// TwinCAT 3 PLC project Untitled1
// ProgramVersion: 3.1.4024.0
// libraries:
//   Tc2_MC2, * (Beckhoff Automation GmbH)
//   Tc2_Standard, * (Beckhoff Automation GmbH)
//   Tc2_System, * (Beckhoff Automation GmbH)
//   Tc3_Module, * (Beckhoff Automation GmbH)
// project tree:
//   Error/DUTs/ E_ErrorPriority.TcDUT, ST_Error.TcDUT
//   Error/GVLs/ Param_Error.TcGVL
//   Error/POUs/ F_ClearError.TcPOU, F_ResetErrorList.TcPOU
//   PermIntlk/PermIntlk/ FB_PermIntlk.TcPOU, GVL_PermIntlk.TcGVL, ITF_PermIntlk.TcIO, Param_PermIntlk.TcGVL, ST_PermIntlkIndex.TcDUT
//   / PlcTask.TcTTO
//   POUs/ MAIN.TcPOU (not stored)
//   Servo/DUTs/ E_ServoTypeMoves.TcDUT, ST_ServoAxisMove.TcDUT (not stored), ST_ServoConfiguration.TcDUT (not stored), ST_ServoInterlocks.TcDUT, ST_ServoMove.TcDUT, ST_ServoStatus.TcDUT
//   Servo/ FB_Servo.TcPOU (not stored), ITF_Servo.TcIO (not stored)
//   Servo/GVLs/ Param_Servo.TcGVL
// real-time tasks:
//   TASK PlcTask: cycle T#10ms, priority 20, ADS port 350
// motion (NC):
//   TASK NC-Task 1 SAF: cycle T#2ms, priority 4, ADS port 501
//   TASK NC-Task 1 SVB: cycle T#10ms, priority 8, ADS port 511
//   AXIS Axis 1 (id 1)
//     OtherSettings: AllowMotionCmdToSlave=true
//     encoder EncType=1
//     drive DrvType=5
//       Analog: TorqueSetpointScale=10, ScaleFactorActTorque=0.1
//       TimeComp: TaskDelayCycles=1
//     controller CtrType=1
//       CtrPara: PriorControlFactor=1
//         Observer: BandWidth=20
// variable links:
//   Untitled1/Untitled1 Instance <-> NC-Task 1 SAF/Axes/Axis 1
//     PlcTask Inputs/MAIN.Servo.Axis.NcToPlc <-> Outputs/ToPlc
//     PlcTask Outputs/MAIN.Servo.Axis.PlcToNc <-> Inputs/FromPlc

CONFIGURATION Untitled1
    RESOURCE PLC ON TwinCAT3
        TASK PlcTask(INTERVAL := T#10ms, PRIORITY := 20);
        PROGRAM MAIN WITH PlcTask : MAIN;
    END_RESOURCE
END_CONFIGURATION

// ---- Error/DUTs/E_ErrorPriority.TcDUT
{attribute 'qualified_only'}
{attribute 'strict'}
TYPE E_ErrorPriority :
(
	Diagnostic := 0,
	Low := 1,
	Medium := 2,
	High := 3,
	Critical := 4
);
END_TYPE

// ---- Error/DUTs/ST_Error.TcDUT
TYPE ST_Error :
STRUCT
	Active : BOOL := FALSE;
	Label : STRING(Param_Error.LABEL_LEN);
	Message : STRING(Param_Error.MESSAGE_LEN);
	Priority : E_ErrorPriority := E_ErrorPriority.Diagnostic;
END_STRUCT
END_TYPE

// ---- PermIntlk/PermIntlk/ST_PermIntlkIndex.TcDUT
TYPE ST_PermIntlkIndex :
STRUCT
	Condition : BOOL := TRUE;
	Description : STRING(Param_PermIntlk.DESCRIPTION_LEN);
END_STRUCT
END_TYPE

// ---- Servo/DUTs/E_ServoTypeMoves.TcDUT
{attribute 'qualified_only'}
{attribute 'strict'}
TYPE E_ServoTypeMoves :
(
	AbsoluteMove := 0,
	RelativeMove := 1,
	VelocityMove := 2,
	DynamicGear  := 3
);
END_TYPE

// ---- Servo/DUTs/ST_ServoInterlocks.TcDUT
TYPE ST_ServoInterlocks :
STRUCT
	Move_Positive : BOOL;
	Move_Negative : BOOL;
	SafetyOk     : BOOL;
	
END_STRUCT
END_TYPE

// ---- Servo/DUTs/ST_ServoMove.TcDUT
TYPE ST_ServoMove :
STRUCT
	Name : STRING(Param_Servo.DESCRIPTION_LEN) := 'Actuator'; //Name visualized on UI
	AdvanceFeedback_Used : BOOL;      //TRUE if advanced state feedback is used  
	RetractFeedback_Used  : BOOL;      //TRUE if retracted state feedback is used  
	AdvanceFeedbackTimeoutError : TIME; // How long we wait to see advanced feedback before we raise timeout error; 0 if not used
	RetractFeedbackTimeoutError : TIME; // How long we wait to see retracted feedback before we raise timeout error; 0 if not used
	SimFeedback_Advance_TimeElapsed : TIME; //If we do not use Advanced Feedback, serves as simulation delay after Advance Output is Set
	SimFeedback_Retract_TimeElapsed : TIME; //If we do not use Retracted Feedback, serves as simulation delay after Advance Output is Set
END_STRUCT
END_TYPE

// ---- Servo/DUTs/ST_ServoStatus.TcDUT
TYPE ST_ServoStatus :
STRUCT
	
	//Status : AXIS_REF.Status;

END_STRUCT
END_TYPE

// ---- Error/GVLs/Param_Error.TcGVL
{attribute 'qualified_only'}
VAR_GLOBAL CONSTANT
	LABEL_LEN : USINT := 40;
	MESSAGE_LEN : USINT := 255;
END_VAR

// ---- PermIntlk/PermIntlk/GVL_PermIntlk.TcGVL
{attribute 'qualified_only'}
{attribute 'global_init_slot' := '49991'}
VAR_GLOBAL CONSTANT
	EMPTY_INDICES : ARRAY[0..(Param_PermIntlk.ARRAY_SIZE-1)] OF ST_PermIntlkIndex := [(Param_Permintlk.ARRAY_SIZE -1)((Condition := TRUE, Description := ''))];
END_VAR

// ---- PermIntlk/PermIntlk/Param_PermIntlk.TcGVL
{attribute 'qualified_only'}
{attribute 'global_init_slot := '49990'}
VAR_GLOBAL CONSTANT
	ARRAY_SIZE : USINT := 16;
	DESCRIPTION_LEN : USINT := 40;
	MESSAGE_LEN : USINT := 127;
END_VAR

// ---- Servo/GVLs/Param_Servo.TcGVL
{attribute 'qualified_only'}
VAR_GLOBAL CONSTANT
	BRANCH_ARRAY_SIZE : USINT := 16;
	DESCRIPTION_LEN : USINT := 40;
	MESSAGE_LEN : UDINT := 255;
	TIMEOUT_LABEL : STRING(Param_Error.LABEL_LEN) := 'Step Timeout';
	TIMEOUT_PRIORITY : E_ErrorPriority := E_ErrorPriority.HIGH;
END_VAR

// ---- PermIntlk/PermIntlk/ITF_PermIntlk.TcIO
INTERFACE ITF_PermIntlk

METHOD M_ClearAll : BOOL
VAR_INPUT
END_VAR
END_METHOD

METHOD M_Set : BOOL
VAR_INPUT
	Index : USINT;
	Description : STRING(Param_PermIntlk.DESCRIPTION_LEN);
	Condition : BOOL;
END_VAR
END_METHOD

{attribute 'monitoring' := 'call'}
PROPERTY P_Message : STRING(Param_PermIntlk.MESSAGE_LEn)
GET
END_GET
END_PROPERTY

{attribute 'monitoring' := 'call'}
PROPERTY P_Name : STRING(Param_PermIntlk.DESCRIPTION_LEN)
GET
END_GET
SET
END_SET
END_PROPERTY

{attribute 'monitoring' := 'call'}
PROPERTY P_OK : BOOL
GET
END_GET
END_PROPERTY

END_INTERFACE

// ---- Error/POUs/F_ClearError.TcPOU
FUNCTION F_ClearError 
VAR_INPUT
	Error : REFERENCE TO ST_Error;
END_VAR
VAR
END_VAR

IF __ISVALIDREF(Error) THEN 
	Error.Active := FALSE;
	Error.Label := '';
	Error.Message := '';
	Error.Priority := E_ErrorPriority.Diagnostic;
END_IF

END_FUNCTION

// ---- Error/POUs/F_ResetErrorList.TcPOU
FUNCTION F_ResetErrorList 
VAR_INPUT
	FirstElement : POINTER TO ST_Error;
	NumElements : UDINT;
END_VAR
VAR
	i : UDINT;
	Instance : POINTER TO ST_Error;
END_VAR

IF FirstElement = 0 THEN 
	RETURN;
END_IF


FOR i := 0 TO (NUMElements - 1) BY 1 DO
	Instance := FirstElement + (i*SIZEOF(firstelement^));
	Instance^.Active := FALSE;
END_FOR

END_FUNCTION

// ---- PermIntlk/PermIntlk/FB_PermIntlk.TcPOU
FUNCTION_BLOCK FB_PermIntlk IMPLEMENTS ITF_PermIntlk

VAR
	Name : STRING(Param_PermIntlk.DESCRIPTION_LEN) := 'Permintlk Name';
	Indices : ARRAY[0..(Param_Permintlk.ARRAY_SIZE-1)] OF ST_PermintlkIndex;
	OK : BOOL;
	Message : STRING(Param_PermIntlk.MESSAGE_LEN);
	
	i : USINT;
END_VAR

OK := TRUE;
Message := '';

FOR i :=0 TO (Param_Permintlk.ARRAY_SIZE-1) BY 1 DO 
	IF NOT Indices[i].Condition THEN 
		OK := FALSE;
		IF Message = '' THEN 
			Message := Indices[i].Description;
		ELSE
			Message := CONCAT(CONCAT(Message, ', '),Indices[i].Description);
		END_IF
	END_IF
END_FOR

METHOD M_ClearAll : BOOL
Indices := GVL_PermIntlk.EMPTY_INDICES;
END_METHOD

METHOD M_Set : BOOL
VAR_INPUT
	Index : USINT;
	Description : STRING(Param_PermIntlk.DESCRIPTION_LEN);
	Condition : BOOL;
END_VAR
IF Index < Param_PermIntlk.ARRAY_SIZE THEN 
	Indices[Index].Description := Description;
	Indices[Index].Condition := Condition;
END_IF
END_METHOD

PROPERTY P_Message : STRING(Param_PermIntlk.MESSAGE_LEn)
GET
P_Message := Message;
END_GET
END_PROPERTY

PROPERTY P_Name : STRING(Param_PermIntlk.DESCRIPTION_LEN)
GET
P_Name := Name;
END_GET
SET
Name := P_Name;
END_SET
END_PROPERTY

PROPERTY P_OK : BOOL
GET
P_OK := OK;
END_GET
END_PROPERTY

END_FUNCTION_BLOCK
